Staubli VAL3: getRow.pgx

program getRow(num& x_nRow[] (dimensions=1), num& x_nMatrix[] (dimensions=2), num x_nRowIndex (dimensions=1))
  local num j
begin
  for j=0 to size(x_nMatrix,2)-1
    x_nRow[j]=x_nMatrix[x_nRowIndex,j]
  endFor
end
